// LS Electric XG5000 project: ESP32_Yellow_detector
// PLC LSPLC

PROGRAM NewProgram (task: 스캔 프로그램)

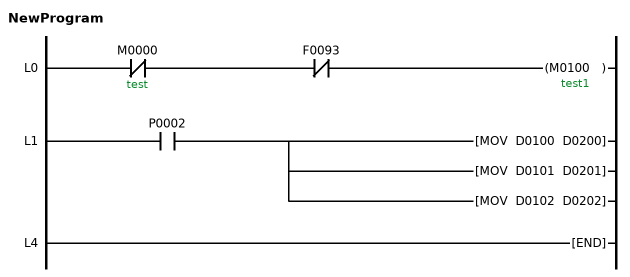
; L0
LOAD NOT  M0000	// test
AND NOT   F0093
OUT       M0100	// test1
; L1
LOAD      P0002
MOV       D0100 D0200
MOV       D0101 D0201
MOV       D0102 D0202
; L4
END